{region '#Template'}
	{attribute 'Category' := 'Universal'}
	{attribute 'Version' := '0.0.1.0'}
	{attribute 'Tags' := 'Universal, Sensor, AI'}
	{attribute 'Description' := 'AI	ohne IO // AI without IO'}
{endregion}
FUNCTION_BLOCK FB_BA_SensorAnalog EXTENDS FB_BA_View
VAR_INPUT
	fVal					: REAL;
END_VAR
VAR_INPUT CONSTANT
	MV						: FB_BA_AI;		
END_VAR
VAR_OUTPUT
	fPresentValue			: REAL;
	bEvent					: BOOL;
	eEventState				: E_BA_EventState;	
END_VAR
VAR
END_VAR

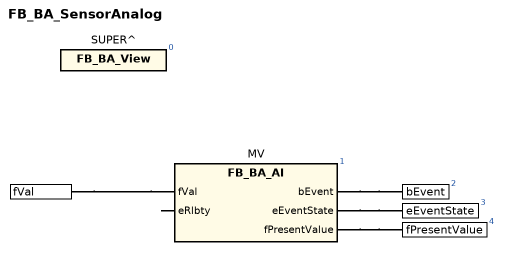
SUPER^(); // FB_BA_View
MV(fVal := fVal); // FB_BA_AI
bEvent := MV.bEvent;
eEventState := MV.eEventState;
fPresentValue := MV.fPresentValue;

METHOD FB_init : BOOL
VAR_INPUT
	bInitRetains : BOOL; // if TRUE, the retain variables are initialized (warm start / cold start)
	bInCopyCode : BOOL;  // if TRUE, the instance afterwards gets moved into the copy code (online change)
END_VAR
MV.iParent						:= THIS^;		
MV.iLabel 						:= LblUniFieldDevice.SensorAnalog_MV;
MV.sObjectName					:= '{Idx=01}';
MV.sDeviceType					:= '';
MV.bEnOutOfService				:= FALSE;
MV.eUnit						:= E_BA_Unit.eTemperature_DegreesCelsius;
MV.fResolution 					:= 0.01;
MV.fScaleOffset 				:= 0; 	
MV.fCOVIncrement				:= BA2_Param.fDefCOVIncrement;
MV.nEventClassID				:= EventClasses.AlarmTechnicalExtended;
MV.stTimeDelay.nToNormal		:= BA2_Param.nDefTimeDelay_ToNormal;
MV.stTimeDelay.nToAbnormal		:= BA2_Param.nDefTimeDelay_ToAbnormal;
MV.stHighLimit.bEnable			:= FALSE;
MV.stHighLimit.fValue			:= 0.0;		
MV.stLowLimit.bEnable			:= FALSE;
MV.stLowLimit.fValue			:= 0.0;
MV.fLimitDeadband 				:= BA2_Param.fDefLimitDeadband;
MV.bAcknowledgeRm				:= FALSE;	
MV.aEventTransitionText[1]		:= Texts.txtExceeded;
MV.aEventTransitionText[2]		:= Texts.txtDisturb;
MV.aEventTransitionText[3]		:= Texts.txtNormal;
MV.bEventDetectionEnable		:= FALSE;
MV.eEnPlantLock					:= E_BA_LockPriority.eNoLock;
END_METHOD

END_FUNCTION_BLOCK

(* stored: Version 1.1.0.1, ProductVersion 3.1.4024.6
   POU FB_BA_SensorAnalog: Id {0a0ed6d5-034f-43e7-9185-6a143a7f098a}, SpecialFunc None
   Method FB_init: Id {a6e402cc-5aee-4b3c-9df2-e05903bbe2ed} *)
